FUNCTION FC_PRG1 : BOOL
VAR_INPUT
	SafetyOK : BOOL;
	KukaStatus : INT;
END_VAR
VAR

	Foutcode : INT; 
	Melding : STRING[20];
END_VAR




CASE DB_PRG1.PRG1Stap OF
	
	0:
		IF SafetyOK AND KukaStatus = 1 AND GVL.b_StartPRG THEN
			DB_PRG1.PRG1Stap := 5;
		END_IF

	5:
		//extruder start aan
		DB_PRG1.t_prgT1_extruderRelaisAan(IN:=TRUE,PT:=T#2S);
		DB10_Alias.qx_relaisExtruderStart := TRUE;
		
		IF DB_PRG1.t_prgT1_extruderRelaisAan.Q THEN
			DB10_Alias.qx_relaisExtruderStart := FALSE;
			DB_PRG1.t_prgT1_extruderRelaisAan.IN := FALSE;
			DB_PRG1.PRG1Stap := 10;
		END_IF
		
	;
	10: // inlezen fotocel lengte
	
		IF DB10_Alias.ix_lengteFC THEN
			DB_PRG1.PRG1Stap := 20;
		END_IF
		
	
	;
	20: // extruder stop aan bij fotocel
	
		DB10_Alias.qx_relaisExtruderStop := TRUE;
		DB_PRG1.PRG1Stap := 30;
		
	;
	
	30:	// cuttingtool aan en extruderstop laag
		DB10_Alias.qx_relaisCuttingtoolActiveer := TRUE;
		DB_PRG1.t_prgT2_extruderRelaisStop(IN:=TRUE,PT:=T#6S); // 4 seconden timeout voor cuttingtool.
		
		IF DB10_Alias.ix_reedCuttingtoolCilinderGesloten THEN
	
			DB10_Alias.qx_relaisExtruderStop := FALSE;
			DB10_Alias.qx_relaisCuttingtoolActiveer := FALSE;
			DB_PRG1.PRG1Stap:= 40;
		(*ELSIF DB_PRG1.t_prgT2.ET > T#2S THEN
			DB10_Alias.qx_relaisExtruderStop := FALSE;
			DB10_Alias.qx_relaisCuttingtoolActiveer := FALSE;
			DB_PRG1.t_prgT2.IN := FALSE;			*)
		ELSIF DB_PRG1.t_prgT2_extruderRelaisStop.Q THEN
			
			DB_PRG1.t_prgT2_extruderRelaisStop.IN := FALSE;
			Foutcode := 1;
			DB_PRG1.PRG1Stap:= 808;
			
		END_IF
	;
	40:	// cuttingtool deactiveer
		
		DB10_Alias.qx_relaisCuttingtoolDeactiveer := TRUE;	
		DB_PRG1.t_prgT2_extruderRelaisStop.IN := FALSE;
		
		DB_PRG1.t_prgT3_cuttingRelaisAan(IN:=TRUE,PT:=T#6S);
		
		IF DB10_Alias.ix_reedCuttingtoolCilinderOpen THEN
			DB10_Alias.qx_relaisCuttingtoolDeactiveer := FALSE;
			GVL.b_startBeweging := TRUE;
			DB_PRG1.PRG1Stap := 50;
			
		ELSIF DB_PRG1.t_prgT3_cuttingRelaisAan.Q THEN
	
			DB_PRG1.t_prgT3_cuttingRelaisAan.IN := FALSE;
			Foutcode := 2;
			DB_PRG1.PRG1Stap:= 808;
			
		END_IF
	
	50: // Check gripperFC en activeer ventiel.
		IF GVL.i_KUKAStatus = 1 THEN
			
			DB10_Alias.qx_ventielEen := TRUE;
			DB_PRG1.t_prgT5_resetKukaGereed(IN := TRUE,PT:=T#3S);
			DB_PRG1.PRG1Stap := 60;
			
		END_IF
	;
	60:	// Timers zijn ter simulatie. Signalen komen vanaf de KUKA
		DB_PRG1.t_prgT5_resetKukaGereed(IN := TRUE,PT:=T#3S);
		DB_PRG1.t_prgT6_Stap60advance(IN := TRUE,PT:=T#20S);
		IF DB_PRG1.t_prgT5_resetKukaGereed.Q THEN 
			DB_PRG1.t_prgT5_resetKukaGereed(IN := FALSE);
			DB10_Alias.ix_kukaGereed := FALSE; /// <<<<<<<<<<<<<<<<< Ter simulatie. Moet vanaf de Kuka komen.
		END_IF;
		IF DB_PRG1.t_prgT6_Stap60advance.Q AND DB10_Alias.ix_kukaGereed THEN
			DB_PRG1.PRG1Stap := 70;
		END_IF
		
		
		

 
	;
	
	808: // Fout fout hella fout
		
		CASE Foutcode OF
			1: Melding := 'Cuttingtool sluiten fout';
			; 
			2: Melding := 'Cuttingtool openen fout';
			;
			3:
			;
			ELSE
			//DB_PRG1.PRG1Stap := 900;	
			
		END_CASE
			IF GVL.safetyOK THEN
				DB_PRG1.PRG1Stap := 900;
			END_IF 			
	;
	900: // reset en terug naar start.
	
		DB_PRG1.t_prgT7_PRGStopRelaisTimer(IN := TRUE,PT:=T#4S);
		DB10_Alias.qx_relaisCuttingtoolDeactiveer := TRUE;
		DB10_Alias.qx_relaisExtruderStop := TRUE;
		DB10_Alias.qx_ventielEen := FALSE;
		
		IF DB_PRG1.t_prgT7_PRGStopRelaisTimer.Q THEN
			DB10_Alias.qx_relaisCuttingtoolDeactiveer := FALSE;
			DB10_Alias.qx_relaisExtruderStop := FALSE;
			DB_PRG1.t_prgT7_PRGStopRelaisTimer.IN := FALSE;
			DB_PRG1.PRG1Stap := 0;
		END_IF
	;
	
	950: // tussentijdse reset of Safety

		
	;
END_CASE

END_FUNCTION

(* stored: Version 1.1.0.1, ProductVersion 3.1.4024.12
   POU FC_PRG1: Id {3c2d693e-a12f-40bc-9ef3-094978264baf}, SpecialFunc None *)
